FUNCTION_BLOCK FLASHER4
  (* Standard: 61499-2 *)
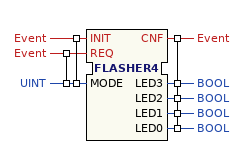
  EVENT_INPUT
    INIT WITH MODE;
    REQ WITH MODE;
  END_EVENT
  EVENT_OUTPUT
    CNF WITH LED3, LED2, LED1, LED0;
  END_EVENT
  VAR_INPUT
    MODE : UINT;
  END_VAR
  VAR_OUTPUT
    LED3 : BOOL;
    LED2 : BOOL;
    LED1 : BOOL;
    LED0 : BOOL;
  END_VAR
  VAR
    OFLO : BOOL;
  END_VAR
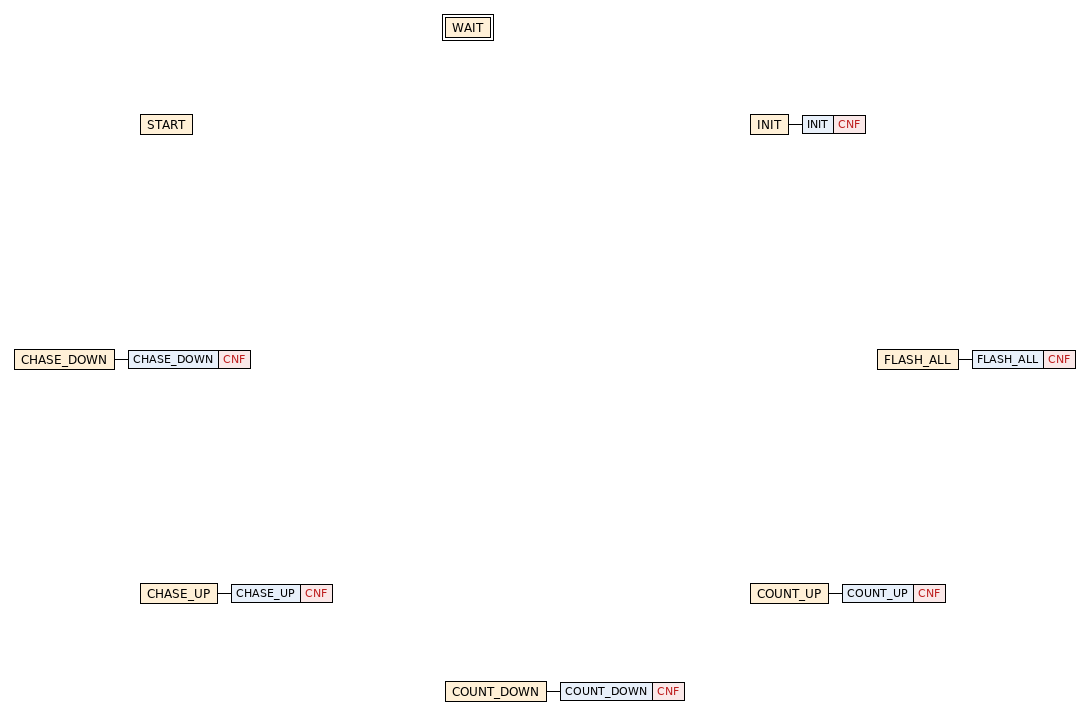
  EC_STATES
    WAIT;
    INIT : INIT -> CNF;
    FLASH_ALL : FLASH_ALL -> CNF;
    COUNT_UP : COUNT_UP -> CNF;
    COUNT_DOWN : COUNT_DOWN -> CNF;
    CHASE_UP : CHASE_UP -> CNF;
    CHASE_DOWN : CHASE_DOWN -> CNF;
    START;
  END_STATES
  EC_TRANSITIONS
    WAIT TO  := INIT;
    WAIT TO  := REQ[MODE = 0];
    WAIT TO  := REQ[MODE = 1];
    WAIT TO  := REQ[MODE = 2];
    WAIT TO  := REQ[MODE = 3];
    WAIT TO  := REQ[MODE = 4];
    INIT TO  := 1;
    FLASH_ALL TO  := 1;
    COUNT_UP TO  := 1;
    COUNT_DOWN TO  := 1;
    CHASE_UP TO  := 1;
    CHASE_DOWN TO  := 1;
    START TO  := 1;
  END_TRANSITIONS
  ALGORITHM INIT IN ST:
LED0 := MODE > 2;&#10;LED1 := 0;&#10;LED2 := 0;&#10;LED3 := 0;&#10;
  END_ALGORITHM
  ALGORITHM COUNT_UP IN ST:
LED0 := NOT LED0;&#10;IF NOT LED0 THEN&#10;  LED1 := NOT LED1;&#10;  IF NOT LED1 THEN&#10;    LED2 := NOT LED2;&#10;    IF NOT LED3 THEN&#10;      LED3 := NOT LED3;&#10;    END_IF;&#10;  END_IF;&#10;END_IF;&#10;
  END_ALGORITHM
  ALGORITHM COUNT_DOWN IN ST:
LED0 := NOT LED0;&#10;IF LED0 THEN&#10;  LED1 := NOT LED1;&#10;  IF LED1 THEN&#10;    LED2 := NOT LED1;&#10;    IF LED2 THEN&#10;      LED3 := NOT LED1;&#10;    END_IF;&#10;  END_IF;&#10;END_IF;&#10;
  END_ALGORITHM
  ALGORITHM FLASH_ALL IN ST:
LED0 := NOT LED0;&#10;LED1 := NOT LED1;&#10;LED2 := NOT LED2;&#10;LED3 := NOT LED3;&#10;
  END_ALGORITHM
  ALGORITHM CHASE_UP IN ST:
OFLO := LED3;&#10;LED3 := LED2;&#10;LED2 := LED1;&#10;LED1 := LED0;&#10;LED0 := OFLO;&#10;
  END_ALGORITHM
  ALGORITHM CHASE_DOWN IN ST:
OFLO := LED0;&#10;LED0 := LED1;&#10;LED1 := LED2;&#10;LED2 := LED3;&#10;LED3 := OFLO;&#10;
  END_ALGORITHM
END_FUNCTION_BLOCK
